// TwinCAT 3 PLC project nepionic_io_test
// ProgramVersion: 3.1.4024.0
// libraries:
//   Tc3_Module, * (Beckhoff Automation GmbH)
//   TcUnit, * (www.tcunit.org)
//   nepionic-io,0.1.0,nepionic
// project tree:
//   Programs/ Main.TcPOU
//   Tasks/ PlcTask.TcTTO
//   Tests/ IO_TestSuite.TcPOU
//   Tests/Mocks/ MockBasicDigitalInput.TcPOU, MockBasicDigitalOutput.TcPOU
// real-time tasks:
//   TASK PlcTask: cycle T#10ms, priority 20, ADS port 350

CONFIGURATION nepionic_io_test
    RESOURCE PLC ON TwinCAT3
        TASK PlcTask(INTERVAL := T#10ms, PRIORITY := 20);
        PROGRAM Main WITH PlcTask : Main;
    END_RESOURCE
END_CONFIGURATION

// ---- Programs/Main.TcPOU
PROGRAM Main
VAR
	io_TestSuite : IO_TestSuite;
END_VAR

TcUnit.Run();

END_PROGRAM

// ---- Tests/IO_TestSuite.TcPOU
FUNCTION_BLOCK PUBLIC IO_TestSuite EXTENDS TcUnit.FB_TestSuite

TestBasicDigitalInput();
TestBasicDigitalOutput();

METHOD PUBLIC TestBasicDigitalInput
VAR
	mockInputRegular : MockBasicDigitalInput(inverted := FALSE);
	mockInputInverted : MockBasicDigitalInput(inverted := TRUE);
END_VAR
Test('TestBasicDigitalInput');

mockInputRegular.MockSetRawInputFalse();

AssertTrue(
	Condition := mockInputRegular.State = FALSE,
	Message := 'State should be FALSE when raw input is FALSE'
);

mockInputRegular.MockSetRawInputTrue();

AssertTrue(
	Condition := mockInputRegular.State = TRUE,
	Message := 'State should be TRUE when raw input is TRUE'
);

mockInputInverted.MockSetRawInputTrue();

AssertTrue(
	Condition := mockInputInverted.State = FALSE,
	Message := 'State should be FALSE when raw input is TRUE and inverted := TRUE'
);

mockInputInverted.MockSetRawInputFalse();

AssertTrue(
	Condition := mockInputInverted.State = TRUE,
	Message := 'State should be TRUE when raw input is FALSE and inverted := TRUE'
);

Test_Finished();
END_METHOD

METHOD PUBLIC TestBasicDigitalOutput
VAR
	mockOutputRegular : MockBasicDigitalOutput(inverted := FALSE);
	mockOutputInverted : MockBasicDigitalOutput(inverted := TRUE);
END_VAR
Test('TestBasicDigitalInput');

mockOutputRegular.State := FALSE;

AssertTrue(
	Condition := mockOutputRegular.RawOutput = FALSE,
	Message := 'raw output should be FALSE when State is FALSE'
);

mockOutputRegular.State := TRUE;

AssertTrue(
	Condition := mockOutputRegular.RawOutput = TRUE,
	Message := 'raw output should be TRUE when State is TRUE'
);

mockOutputInverted.State := FALSE;

AssertTrue(
	Condition := mockOutputInverted.RawOutput = TRUE,
	Message := 'raw output should be TRUE when State is FALSE and inverted := TRUE'
);

mockOutputInverted.State := TRUE;

AssertTrue(
	Condition := mockOutputInverted.RawOutput = FALSE,
	Message := 'raw output should be TRUE when State is FALSE and inverted := TRUE'
);

Test_Finished();
END_METHOD

END_FUNCTION_BLOCK

// ---- Tests/Mocks/MockBasicDigitalInput.TcPOU
{attribute 'linkalways'} 
{attribute 'no_explicit_call' := 'This FB is a CLASS and must be accessed using methods or properties'}
{attribute 'enable_dynamic_creation'}
FUNCTION_BLOCK MockBasicDigitalInput EXTENDS BasicDigitalInput

METHOD MockSetRawInputFalse : BOOL
SUPER^.input := FALSE;
END_METHOD

METHOD MockSetRawInputTrue : BOOL
SUPER^.input := TRUE;
END_METHOD

END_FUNCTION_BLOCK

// ---- Tests/Mocks/MockBasicDigitalOutput.TcPOU
{attribute 'linkalways'} 
{attribute 'no_explicit_call' := 'This FB is a CLASS and must be accessed using methods or properties'}
{attribute 'enable_dynamic_creation'}
FUNCTION_BLOCK MockBasicDigitalOutput EXTENDS BasicDigitalOutput

PROPERTY RawOutput : BOOL
GET
RawOutput := SUPER^.output;
END_GET
END_PROPERTY

END_FUNCTION_BLOCK
